FUNCTION_BLOCK E_CALIBRATE (* Calibrate allows for offset and scale calibration of an analog input. *)
  (* Standard: 61499-1; Description: version 1.3	11. mar. 2009 programmer 	hugo tested BY		hans Calibrate allows for offset and scale calibration of an analog input. offset is calibrated to a stored reference Y_offset while CO is true. after the offset is calibrated, scale can be calibrated to a reference value Y_scale while CS is true. *)
  (* Version 1.0, 2026-05-06, franz *)
  PACKAGE OSCAT::Basic::POUs::Engineering::measurements;
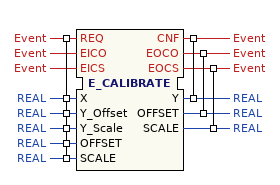
  EVENT_INPUT
    REQ WITH X, Y_Offset, Y_Scale, OFFSET, SCALE; (* Normal Execution Request *)
    EICO; (* Calibrate Offset *)
    EICS; (* Calibrate Scale *)
  END_EVENT
  EVENT_OUTPUT
    CNF WITH Y; (* Execution Confirmation *)
    EOCO WITH OFFSET; (* Calibrate Offset *)
    EOCS WITH SCALE; (* Calibrate Scale *)
  END_EVENT
  VAR_INPUT
    X : REAL; (* Input *)
    Y_Offset : REAL; (* Reference for offset calibration *)
    Y_Scale : REAL; (* Reference for scale calibration *)
  END_VAR
  VAR_OUTPUT
    Y : REAL; (* Calibrated Output *)
  END_VAR
  VAR_IN_OUT
    OFFSET : REAL := 0.0; (* Offset value *)
    SCALE : REAL := 1.0; (* Scale value *)
  END_VAR
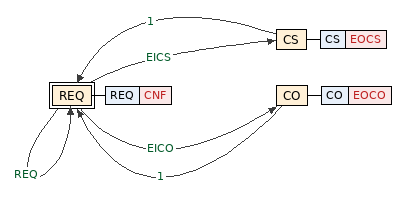
  EC_STATES
    REQ : REQ -> CNF;
    CO : CO -> EOCO;
    CS : CS -> EOCS;
  END_STATES
  EC_TRANSITIONS
    REQ TO CS := EICS;
    REQ TO CO := EICO;
    CS TO REQ := 1;
    CO TO REQ := 1;
    REQ TO REQ := REQ;
  END_TRANSITIONS
  ALGORITHM REQ IN ST:
(* calculate output *)
Y := (X + OFFSET) * SCALE;

(* revision history hm 22.2.2007 rev 1.2 changed VAR RETAIN PERSISTENT to VAR RETAIN for better
 * compatibility wago lon contollers do not support persisitent
 * *
 * hm	11. mar. 2009	rev 1.3 changed real constants to use dot syntax *)
  END_ALGORITHM
  ALGORITHM CO IN ST:
OFFSET := Y_Offset - X;
  END_ALGORITHM
  ALGORITHM CS IN ST:
SCALE := Y_Scale / (X + OFFSET);
  END_ALGORITHM
END_FUNCTION_BLOCK
